TYPE PickerComSubscribe :
STRUCT
  Request : PickerComRequest; // contains booleans that are used to start a specific sequence.
  Equipment : PickerComSubscribeEquipment;  // structs for equipment objects which are used by the bridges
END_STRUCT
END_TYPE

(* stored: Version 1.1.0.1
   DUT PickerComSubscribe: Id {01459558-85e9-4ef9-bfb8-8961108ec7b4} *)
